{attribute 'contextName':='ComTask'}
PROGRAM SerialBackCom
VAR
	i : USINT;
END_VAR

FOR i:= 1 TO GVL_RS232.cNoOfSerialPorts BY 1 DO
	IF GVL_RS232.aSerialPorts[i] > 0 THEN
		GVL_RS232.aSerialPorts[i]^();	
	END_IF
END_FOR

END_PROGRAM

(* stored: Version 1.1.0.1, ProductVersion 3.1.4024.6
   POU SerialBackCom: Id {2f0cc4ca-9e34-42ef-8561-eb295bc82e89}, SpecialFunc None *)
